FUNCTION_BLOCK M_INV (* Solve the matrix equation IN1*OUT=IN2 for OUT by inverting IN1 *)
  (* Standard: 61499-1; Classification: Matrix Operations; Function: Addition *)
  (* Version 0.0, 2002-03-06, JHC, Rockwell Automation *)
  (* Compiler header: package fb.rt.math; *)
  (* Compiler classdef: public class M_MUL extends M_ADD *)
  (* Compiler Java IBM VisualAge 3.0 *)
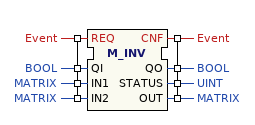
  EVENT_INPUT
    REQ WITH QI, IN1, IN2; (* Solve IN1*OUT=IN2 for OUT *)
  END_EVENT
  EVENT_OUTPUT
    CNF WITH QO, STATUS, OUT; (* Confirmation of Requested Service *)
  END_EVENT
  VAR_INPUT
    QI : BOOL; (* Event Input Qualifier *)
    IN1 : MATRIX;
    IN2 : MATRIX;
  END_VAR
  VAR_OUTPUT
    QO : BOOL; (* Event Output Qualifier *)
    STATUS : UINT; (* Service Status *)
    OUT : MATRIX; (* IN1(inverse)*IN2 *)
  END_VAR
END_FUNCTION_BLOCK
